// TwinCAT 3 PLC project ExampleProject
// ProgramVersion: 3.1.4026.9
// CompilerDefines: VISU_USEWSTRING
// libraries:
//   Tc2_Standard, * (Beckhoff Automation GmbH)
//   Tc2_System, * (Beckhoff Automation GmbH)
//   Core, * (_)
//   Utils, * (_)
// project tree:
//   / GlobalTextList.TcGTLO, PlcTask.TcTTO
//   Heating/Ctx/ Heating_Ctx_Hmi.TcPOU, Heating_Ctx_Io.TcDUT, Heating_Ctx_Priv.TcPOU, Heating_Ctx_States.TcPOU (not stored)
//   Heating/Ctx/Io/ Heating_Ctx_Io_In.TcDUT (not stored), Heating_Ctx_Io_Out.TcDUT (not stored)
//   Heating/ Heating.TcPOU, Heating_Ctx.TcPOU
//   Heating/Receivers/ Heating_PassiveCountRec.TcPOU, Heating_RequestRec.TcPOU
//   Heating/State/ Heating_State.TcPOU (not stored), Heating_State_Enabled.TcPOU, Heating_State_Disabled.TcPOU, Heating_State_Heatup.TcPOU, Heating_State_Pumping.TcPOU, Heating_State_Safety.TcPOU, Heating_State_Fault.TcPOU
//   MAIN/ ArgAsIRoom.TcPOU, CST.TcGVL, COL.TcGVL, MAIN.TcPOU
//   Room/Rooms/FullRoom/ PassiveTempTimeRoomWithMultipleValves.TcPOU, Room_Settings_PassiveTempTime.TcDUT (not stored), PassiveTempTimeRoom.TcPOU
//   Room/Rooms/PassiveRoom/ PassiveRoom.TcPOU
//   Room/Rooms/TempRoom/ Room_Settings_TemperatureSettings.TcDUT, TempRoom.TcPOU, TempRoomWithMultipleSensors.TcPOU
//   Room/Rooms/TimeRoom/ Room_Settings_TimeSettings.TcDUT, TimeRoom.TcPOU
//   Room/Rooms/TempTimeRoom/ Room_Settings_TempTime.TcDUT (not stored), TempTimeRoom.TcPOU
//   Room/Shared Interface/ I_Room.TcIO, RoomInterface.TcPOU (not stored)
//   Room/Ctx/ Room_Ctx_Hmi.TcPOU, Room_Ctx_Io.TcDUT, Room_Ctx_Priv.TcPOU, Room_Ctx_States.TcPOU
//   Room/Receivers/ Room_SystemReceiver.TcPOU
//   Room/Rooms/ AbstractRoom.TcPOU
//   Room/ Room_Ctx.TcPOU
//   Room/State/ Room_State.TcPOU, Room_State_DemandPassive.TcPOU, Room_State_Idle.TcPOU, Room_State_Fault.TcPOU, Room_State_DemandTemperature.TcPOU, Room_State_Disabled.TcPOU, Room_State_DemandTime.TcPOU, Room_State_SystemOff.TcPOU
//   Room/UI/ Room_UiLogic.TcPOU
//   Safety/ Safety.TcPOU, Safety_Hmi.TcPOU

CONFIGURATION ExampleProject
    RESOURCE PLC ON TwinCAT3
        TASK PlcTask(INTERVAL := T#10ms, PRIORITY := 20);
        PROGRAM MAIN WITH PlcTask : MAIN;
    END_RESOURCE
END_CONFIGURATION

// ---- Heating/Ctx/Heating_Ctx_Io.TcDUT
TYPE Heating_Ctx_Io :
STRUCT
	in		: Heating_Ctx_Io_In;
	out		: Heating_Ctx_Io_Out;
END_STRUCT
END_TYPE

// ---- Room/Rooms/TempRoom/Room_Settings_TemperatureSettings.TcDUT
TYPE Room_Settings_TemperatureSettings :
STRUCT
	rLow	: REAL := 19.0;
	rHigh	: REAL := 19.3;
END_STRUCT
END_TYPE

// ---- Room/Rooms/TimeRoom/Room_Settings_TimeSettings.TcDUT
TYPE Room_Settings_TimeSettings :
STRUCT
	nOff		: UDINT := TIME_TO_UDINT(T#30S);
	nOn			: UDINT := TIME_TO_UDINT(T#30S);
END_STRUCT
END_TYPE

// ---- Room/Ctx/Room_Ctx_Io.TcDUT
TYPE Room_Ctx_Io :
STRUCT
	in		: Heating_Ctx_Io_In;
	out		: Heating_Ctx_Io_Out;
END_STRUCT
END_TYPE

// ---- MAIN/CST.TcGVL
{attribute 'qualified_only'}
VAR_GLOBAL CONSTANT
	MAX_PASSIVE_ROOM		: UDINT := 3;
END_VAR

// ---- MAIN/COL.TcGVL
{attribute 'qualified_only'}
VAR_GLOBAL CONSTANT
{warning disable C0228}	// Disable warning: No initial value for variable ...
	RED			: Color(255, 0, 0, 255);
	BLACK		: Color(0, 0, 0, 255);
	ORANGE		: Color(255, 160, 0, 255);
	WHITE		: Color(255, 255, 255, 255);
{warning restore C0228}
END_VAR

// ---- Room/Shared Interface/I_Room.TcIO
INTERFACE I_Room EXTENDS I_Arg

PROPERTY Active : BOOL
GET
END_GET
END_PROPERTY

METHOD Close
END_METHOD

PROPERTY Id : UDINT
GET
END_GET
END_PROPERTY

PROPERTY IsClosed : BOOL
GET
END_GET
END_PROPERTY

PROPERTY IsOpen : BOOL
GET
END_GET
END_PROPERTY

PROPERTY IsReady : BOOL
GET
END_GET
END_PROPERTY

METHOD Open
END_METHOD

PROPERTY Timeout : TIME
GET
END_GET
END_PROPERTY

METHOD TriggerFault
VAR_INPUT
	sErrorText		: Str;
END_VAR
END_METHOD

END_INTERFACE

// ---- MAIN/MAIN.TcPOU
PROGRAM MAIN
VAR
	safety				: Safety<2>;
	heating				: Heating;
	standardRoom		: ARRAY[1..5] OF TempTimeRoom;
	receptionRoom		: PassiveRoom;
	conferentionRoom01	: PassiveTempTimeRoom;
	conferentionRoom02	: PassiveTempTimeRoomWithMultipleValves<3>;
	storeRoom01			: TempRoom;
	storeRoom02			: TempRoomWithMultipleSensors<3>;
	
	bSimulation			: BOOL;
	
	dbgList				: DebugList;	
	
	
	
END_VAR

Runtime();

IF bSimulation THEN
	_Sim();
ELSE
	_IO();	
END_IF

METHOD PRIVATE _IO
END_METHOD

METHOD PRIVATE _Sim
IF safety.bErrAck THEN
	safety.bSafetyOk := TRUE;
END_IF
END_METHOD

END_PROGRAM

// ---- Safety/Safety.TcPOU
FUNCTION_BLOCK Safety 
VAR_GENERIC CONSTANT
	ESTOP_CAP		: UDINT := 2;
END_VAR
IMPLEMENTS I_Execute
VAR_INPUT
	bSafetyOk		: BOOL;
	bEStopActive	: ARRAY[1..ESTOP_CAP] OF BOOL;
END_VAR
VAR_OUTPUT
	bSafetyRun		: BOOL;
	bErrAck			: BOOL;
END_VAR
VAR
	_this			: Entity;
	_ctx			: Heating_Ctx;
	_tag			: Tag('Safety');
	_compTag		: Comp(_tag, _this);
	_exe			: Execute(THIS^);
	
	_onSafetyChange		: Signal;
	_compOnSafetyChange	: Comp(_onSafetyChange, _this);
	
	_bSafetyStopActive	: BoolArg;
	
	_hmi				: Safety_Hmi<ESTOP_CAP>;
	
	_nStep				: USINT;
	_tonTimeout			: TON;
END_VAR

METHOD Execute
VAR
	i			: UDINT;
END_VAR
FOR i := 1 TO ESTOP_CAP DO
	_hmi.bEStopActive[i] := bESTopActive[i];
END_FOR


CASE _nStep OF
	0: // Fault Init
		_bSafetyStopActive.Val := TRUE;
		_onSafetyChange.Emit(_bSafetyStopActive);
		bSafetyRun	:= FALSE;
		
		_nStep := 1;
		
		_hmi.bHideReset := FALSE;
		_hmi.nStatusColor := COL.RED.Raw;
		_hmi.sStatusText := 'Safety Stop Activated!';

	1: // Fault
		IF bSafetyOk AND _hmi.bReset THEN
			_hmi.bReset := FALSE;
			
			_nStep := 2;
		END_IF

	2: // Reset init
		bSafetyRun	:= TRUE;
		
		_nStep		:= 3;
		
		_hmi.bHideReset := FALSE;
		_hmi.nStatusColor := COL.RED.Raw;
		_hmi.sStatusText := 'Reset in progress...';
		
	3: // Reset
	
		bErrAck		:= TRUE;
		
		_tonTimeout(IN := TRUE, PT := T#5S);
		
		IF bSafetyOk THEN
			_tonTimeout(IN := FALSE);
			_nStep := 4;
		ELSIF _tonTimeout.Q THEN
			_tonTimeout(IN := FALSE);
			_nStep := 0;
		END_IF	

	4:	// Op Init
		bErrAck		:= FALSE;
	
		_bSafetyStopActive.Val := FALSE;
		_onSafetyChange.Emit(_bSafetyStopActive);
		_nStep := 5;
		
		_hmi.bHideReset := FALSE;
		_hmi.nStatusColor := COL.BLACK.Raw;
		_hmi.sStatusText := 'Safety OK!';

	5:	// Op
		IF NOT bSafetyOk THEN
			_nStep := 0;
		END_IF


		
END_CASE
END_METHOD

END_FUNCTION_BLOCK

// ---- Heating/Heating_Ctx.TcPOU
FUNCTION_BLOCK Heating_Ctx
VAR_INPUT
	io		: Heating_Ctx_Io;
	hmi		: Heating_Ctx_Hmi;
	state	: Heating_Ctx_States;
	priv	: Heating_Ctx_Priv;
END_VAR

END_FUNCTION_BLOCK

// ---- Heating/Ctx/Heating_Ctx_Hmi.TcPOU
FUNCTION_BLOCK Heating_Ctx_Hmi
VAR_INPUT
	sStatusText				: Str;
	nStatusColor			: LWORD;
	
	bButton					: BOOL;
	sButtonText				: Str;
	nButtonColor			: LWORD;	
END_VAR

END_FUNCTION_BLOCK

// ---- Heating/Ctx/Heating_Ctx_Priv.TcPOU
FUNCTION_BLOCK Heating_Ctx_Priv
VAR_INPUT
	iActiveRoom		: I_Arg;
	nPassiveRooms	: UDINT;	
END_VAR
VAR_OUTPUT
	iOnEnable		: I_SignalEmit;
	iOnDisable		: I_SignalEmit;
	iOnPause		: I_SignalEmit;
	iOnResume		: I_SignalEmit;
	
	iQueue			: I_MutArgQueue;
END_VAR

END_FUNCTION_BLOCK

// ---- Safety/Safety_Hmi.TcPOU
FUNCTION_BLOCK Safety_Hmi
VAR_GENERIC CONSTANT
	ESTOP_CAP		: UDINT := 4;
END_VAR

VAR_INPUT
	bEStopActive	: ARRAY[1..ESTOP_CAP] OF BOOL;
	
	sStatusText		: Str;
	nStatusColor	: LWORD;
	
	bReset			: BOOL;
	bHideReset		: BOOL;
END_VAR

END_FUNCTION_BLOCK

// ---- Heating/Heating.TcPOU
FUNCTION_BLOCK Heating IMPLEMENTS I_Execute
VAR_INPUT
	bPumpOverload	: BOOL;
	bBurnerOverload	: BOOL;

	rBoilerTemp		: REAL;
	rBoilerPressure	: REAL;	
END_VAR
VAR_OUTPUT
	bPump			: BOOL;
	bBurner			: BOOL;
END_VAR
VAR
	_this			: Entity;
	_ctx			: Heating_Ctx;
	_tag			: Tag('Heating');
	_compTag		: Comp(_tag, _this);
	_exe			: Execute(THIS^);
	
	_onEnable		: Signal;
	_compOnEnable	: Comp(_onEnable, _this);
	_proxOnEnable	: SignalProxy(_onEnable, _ctx.priv.iOnEnable);
	
	_onDisable		: Signal;
	_compOnDisable	: Comp(_onDisable, _this);
	_proxOnDisable	: SignalProxy(_onDisable, _ctx.priv.iOnDisable);
	
	_onPause		: Signal;
	_compOnPause	: Comp(_onPause, _this);
	_proxOnPause	: SignalProxy(_onPause, _ctx.priv.iOnPause);
	
	_onResume		: Signal;
	_compOnResume	: Comp(_onResume, _this);
	_proxOnResume	: SignalProxy(_onResume, _ctx.priv.iOnResume);
	
	_smgr			: StateManager<6>(_this);
	_proxSmgr		: StateManagerProxy(_smgr, _ctx.state.iMgr);
	
	_disabled		: Heating_State_Disabled(_this, _ctx);
	_proxDisabled	: StateProxy(_disabled, _ctx.state.iDisable);
	
	_safety			: Heating_State_Safety(_this, _ctx);
	_proxSafety		: StateProxy(_safety, _ctx.state.iSafety);
	
	_fault			: Heating_State_Fault(_this, _ctx);
	_proxFault		: StateProxy(_fault, _ctx.state.iFault);
	
	_enabled		: Heating_State_Enabled(_this, _ctx);
	_proxEnabled	: StateProxy(_enabled, _ctx.state.iEnable);
	
	_pumping		: Heating_State_Pumping(_this, _ctx);
	_proxPumping	: StateProxy(_pumping, _ctx.state.iPump);
	
	_heatup			: Heating_State_Heatup(_this, _ctx);
	_proxHeatup		: StateProxy(_heatup, _ctx.state.iHeatup);

	_passiveHeatingCount		: Heating_PassiveCountRec(_ctx);
	_passiveHeatingCountRec		: Receiver(_passiveHeatingCount);
	_compPassiveHeatingCountRec	: Comp(_passiveHeatingCountRec, _this);
	
	_request					: Heating_RequestRec(_ctx);
	_requestRec					: Receiver(_request);
	_compRequestRec				: Comp(_requestRec, _this);
	
	_queue						: ArgQueue<CST.MAX_ROOM>;
	_queueProxy					: ArgQueueProxy(_queue, _ctx.priv.iQueue);
	
	_tonPump	: TON;
	_tonBurner	: TON;
END_VAR

METHOD Execute
// Inputs
_ctx.io.in.bBurnerOverload := bBurnerOverload;
_ctx.io.in.bPumpOverload := bPumpOverload;
_ctx.io.in.rBoilerPressure := rBoilerPressure;
_ctx.io.in.rBoilerTemp := rBoilerTemp;

// Outputs
_tonPump(IN := _ctx.io.out.bPump, PT := T#2S, Q => bPump);
_tonBurner(IN := _ctx.io.out.bBurner, PT := T#2S, Q => bBurner);
END_METHOD

END_FUNCTION_BLOCK

// ---- Heating/State/Heating_State_Disabled.TcPOU
FUNCTION_BLOCK Heating_State_Disabled EXTENDS Heating_State
VAR_INPUT
END_VAR
VAR_OUTPUT
END_VAR
VAR
END_VAR

METHOD OnExecute
IF _ctx.hmi.bButton THEN
	_ctx.hmi.bButton := FALSE;
	_ctx.state.iMgr.Request(_ctx.state.iEnable);
END_IF
END_METHOD

METHOD OnInit
_ctx.hmi.sStatusText := 'Heating disabled!';
_ctx.hmi.nStatusColor := COL.BLACK.Raw;

_ctx.hmi.sButtonText := 'Press to ENABLE!';
_ctx.hmi.nButtonColor := COL.BLACK.Raw;

_ctx.io.out.bBurner := FALSE;
_ctx.io.out.bPump := FALSE;

_ctx.priv.iOnDisable.Emit();
END_METHOD

END_FUNCTION_BLOCK

// ---- Heating/State/Heating_State_Safety.TcPOU
FUNCTION_BLOCK Heating_State_Safety EXTENDS Heating_State IMPLEMENTS I_Callable, I_Init
VAR
	_init					: Init(THIS^);
	_safetyRec				: Receiver(THIS^);
	_bSafetyStopActive			: BOOL;
END_VAR

METHOD Call
VAR_INPUT
	iArg		: Core.I_Arg;
END_VAR
VAR
	_iSafeModeOn: I_BoolArg;
END_VAR
IF IsOk(ArgToIBoolArg(iArg, iVal => _iSafeModeOn)) THEN
	IF _iSafeModeOn.Val THEN
		_bSafetyStopActive := TRUE;
		_ctx.state.iMgr.Request(_ctx.state.iSafety);
	ELSE
		_bSafetyStopActive := FALSE;
		_ctx.state.iMgr.Request(_ctx.state.iDisable);
	END_IF
END_IF
END_METHOD

METHOD CanDeactivate : BOOL
CanDeactivate := NOT _bSafetyStopActive;
END_METHOD

METHOD Init
VAR
	i			: Iter(1);
	_r			: Result;
	
	_iEntity	: I_Entity;
	_iSignal	: I_Signal;
	
	
END_VAR
WHILE IsOk(GetEntity(i.Next(), iEntity => _iEntity)) DO
	IF IsOk(GetSignal(_iEntity, '*.onSafetyChange', iSignal => _iSignal)) THEN
		IF IsErr(_iSignal.Pair(_safetyRec), nOut => _r) THEN
			DebugMsg(_iSignal, CONCAT('Could not be paired! Error code: ', TO_STRING(_r)));
		END_IF
		
		EXIT;
	END_IF
END_WHILE

IF NOT IsOk(_r) THEN
	DebugMsg(THIS^, CONCAT('_safetyRec not paired! Error code: ', TO_STRING(_r)));
END_IF
END_METHOD

METHOD OnInit
_ctx.hmi.sStatusText := 'Safety engaged! Check safety system...';
_ctx.hmi.nStatusColor := COL.RED.Raw;

_ctx.hmi.sButtonText := '';
_ctx.hmi.nButtonColor := COL.INVISIBLE.Raw;

_ctx.io.out.bBurner := FALSE;
_ctx.io.out.bPump := FALSE;

_ctx.priv.iOnDisable.Emit();
END_METHOD

END_FUNCTION_BLOCK

// ---- Heating/State/Heating_State_Fault.TcPOU
FUNCTION_BLOCK Heating_State_Fault EXTENDS Heating_State
VAR_INPUT
END_VAR
VAR_OUTPUT
END_VAR
VAR
END_VAR

METHOD OnInit
_ctx.hmi.sStatusText := 'Heating enabled: Waiting for requests...';
_ctx.hmi.nStatusColor := COL.BLACK.Raw;

_ctx.hmi.sButtonText := 'Press to DISABLE!';
_ctx.hmi.nButtonColor := COL.BLACK.Raw;

_ctx.io.out.bBurner := FALSE;
_ctx.io.out.bPump := FALSE;
END_METHOD

END_FUNCTION_BLOCK

// ---- Heating/State/Heating_State_Enabled.TcPOU
FUNCTION_BLOCK Heating_State_Enabled EXTENDS Heating_State
VAR_INPUT
END_VAR
VAR_OUTPUT
END_VAR
VAR
END_VAR

METHOD OnExecute
VAR
	_iRoomArg		: I_Arg;
END_VAR
IF _ctx.hmi.bButton THEN
	_ctx.hmi.bButton := FALSE;
	_ctx.state.iMgr.Request(_ctx.state.iDisable);
	
ELSIF _ctx.io.in.rBoilerTemp < _ctx.hmi.rMinTemperature THEN
	_ctx.state.iMgr.Request(_ctx.state.iHeatup);
	
ELSIF IsOk(_ctx.priv.iQueue.Pop(iArg => _iRoomArg)) THEN
	IF IsOk(ArgAsIRoom(_iRoomArg, iDest => _ctx.priv.iActiveRoom)) THEN
		_ctx.state.iMgr.Request(_ctx.state.iPump);
	ELSE
		_ctx.hmi.sErrorText := 'Room Queue - Incorrect iRoomArg!';
	END_IF
END_IF

IF NOT _ctx.io.out.bPump AND _ctx.priv.nPassiveRooms <> 0 THEN
	_ctx.io.out.bPump := TRUE;
	_ctx.hmi.sStatusText := 'Heating enabled: Circulating...';
	
ELSIF _ctx.io.out.bPump AND _ctx.priv.nPassiveRooms <> 0 THEN
	_ctx.io.out.bPump := FALSE;
	_ctx.hmi.sStatusText := 'Heating enabled: Waiting for requests...';
	
END_IF
END_METHOD

METHOD OnInit
_ctx.hmi.sStatusText := 'Heating enabled: Waiting for requests...';
_ctx.hmi.nStatusColor := COL.BLACK.Raw;

_ctx.hmi.sButtonText := 'Press to DISABLE!';
_ctx.hmi.nButtonColor := COL.BLACK.Raw;

_ctx.io.out.bBurner := FALSE;
_ctx.io.out.bPump := FALSE;

_ctx.priv.iOnEnable.Emit();
_ctx.priv.iOnResume.Emit();
END_METHOD

END_FUNCTION_BLOCK

// ---- MAIN/ArgAsIRoom.TcPOU
FUNCTION ArgAsIRoom : Result
VAR_INPUT
	iSource	: I_Arg;
END_VAR
VAR_OUTPUT
	iDest	: I_Room;
END_VAR

IF iSource = 0 THEN
	ArgAsIRoom := Err.Itf0;
	RETURN;
END_IF

IF __QUERYINTERFACE(iSource, iDest) THEN
	ArgAsIRoom := Ok;
ELSE
	ArgAsIRoom := Err.NoMatch;
END_IF

END_FUNCTION

// ---- Heating/State/Heating_State_Pumping.TcPOU
FUNCTION_BLOCK Heating_State_Pumping EXTENDS Heating_State
VAR CONSTANT
	ERROR_STEP		: USINT := 8;
	READY_STEP		: USINT := 9;
END_VAR
VAR
	_nStep		: USINT;
	_tonTimeout	: TON;
END_VAR

METHOD CanActivate : BOOL
CanActivate :=  _ctx.state.iMgr.Current = _ctx.state.iEnable;
END_METHOD

METHOD OnExecute
VAR
	strb		: Strb;
END_VAR
_tonTimeout(IN := TRUE);
IF _tonTimeout.Q THEN
	_nStep := ERROR_STEP;
	_ctx.hmi.sErrorText := strb.Append('Pumping - Timeout at step ')
								.Append(USINT_TO_STRING(_nStep))
								.Append('!')
								.Read();
ELSIF _ctx.priv.iActiveRoom = 0 THEN
	_nStep := ERROR_STEP;
	_ctx.hmi.sErrorText := 'Pumping -Incorrect iActiveRoom value!';
ELSIF _ctx.priv.iActiveRoom.Abort THEN
	_nStep := 6;
END_IF

CASE _nStep OF
	0:
		_ctx.priv.iActiveRoom.Open();
		_nStep := 1;
		
	1:
		IF _ctx.priv.iActiveRoom.IsOpen THEN
			_nStep := 2;
		END_IF
	2:	
		_ctx.io.out.bBurner := TRUE;
		_ctx.io.out.bPump := TRUE;
		_nStep := 3;
		
	3:
		_tonTimeout(IN := FALSE);
		IF _ctx.priv.iActiveRoom.IsReady THEN
			_nStep := 4;
		END_IF
	4:	
		_ctx.io.out.bBurner := FALSE;
		_ctx.io.out.bPump := FALSE;
		_nStep := 5;
	5:
		_ctx.priv.iActiveRoom.Close();
		_nStep := 6;
	6:
		IF _ctx.priv.iActiveRoom.IsClosed THEN
			_nStep := 7;
		END_IF
	7:
		_ctx.state.iMgr.Request(_ctx.state.iEnable);
		_nStep := READY_STEP;
	ERROR_STEP:
		_ctx.state.iMgr.Request(_ctx.state.iFault);
		_nStep := READY_STEP;
END_CASE
END_METHOD

METHOD OnInit
VAR
	strb			: Strb;
END_VAR
_ctx.hmi.sStatusText := strb.Append('Heating enabled: Pumping to room ')
							.Append(UDINT_TO_STRING(_ctx.priv.iActiveRoom.Id))
							.Append('...')
							.Read();
							
_ctx.hmi.nStatusColor := COL.BLACK.Raw;

_ctx.hmi.sButtonText := 'Press to DISABLE!';
_ctx.hmi.nButtonColor := COL.BLACK.Raw;

_ctx.io.out.bBurner := FALSE;
_ctx.io.out.bPump := FALSE;

_ctx.priv.iOnPause.Emit();

_nStep := 0;
_tonTimeout(IN := FALSE);
END_METHOD

END_FUNCTION_BLOCK

// ---- Heating/State/Heating_State_Heatup.TcPOU
FUNCTION_BLOCK Heating_State_Heatup EXTENDS Heating_State
VAR_INPUT
END_VAR
VAR_OUTPUT
END_VAR
VAR
END_VAR

METHOD CanActivate : BOOL
CanActivate :=  _ctx.state.iMgr.Current = _ctx.state.iEnable;
END_METHOD

METHOD OnExecute
IF _ctx.hmi.bButton THEN
	_ctx.hmi.bButton := FALSE;
	_ctx.state.iMgr.Request(_ctx.state.iEnable);
END_IF
END_METHOD

METHOD OnInit
_ctx.hmi.sStatusText := 'Heating enabled: Heating up...';
_ctx.hmi.nStatusColor := COL.BLACK.Raw;

_ctx.hmi.sButtonText := 'Press to DISABLE!';
_ctx.hmi.nButtonColor := COL.BLACK.Raw;

_ctx.io.out.bBurner := TRUE;
_ctx.io.out.bPump := TRUE;
END_METHOD

END_FUNCTION_BLOCK

// ---- Heating/Receivers/Heating_PassiveCountRec.TcPOU
FUNCTION_BLOCK Heating_PassiveCountRec IMPLEMENTS I_Callable
VAR
	_ctx			: REFERENCE TO Heating_Ctx;
END_VAR

METHOD Call
VAR_INPUT
	iArg				: Core.I_Arg;
END_VAR
VAR
	_iPassiveHeatingOn	: I_BoolArg;
END_VAR
IF IsOk(ArgToIBoolArg(iArg, iVal => _iPassiveHeatingOn)) THEN
	IF _iPassiveHeatingOn.Val THEN
		IF _ctx.priv.nPassiveRooms > CST.MAX_PASSIVE_ROOM THEN
			_ctx.priv.nPassiveRooms := _ctx.priv.nPassiveRooms + 1;
		END_IF 	
	ELSE
		IF _ctx.priv.nPassiveRooms > 0 THEN
			_ctx.priv.nPassiveRooms := _ctx.priv.nPassiveRooms - 1;
		END_IF
	END_IF
END_IF
END_METHOD

//FB_Init is always available implicitly and it is used primarily for initialization.
//The return value is not evaluated. For a specific influence, you can also declare the
//methods explicitly and provide additional code there with the standard initialization
//code. You can evaluate the return value.
METHOD FB_Init: BOOL
VAR_INPUT
    bInitRetains: BOOL; // TRUE: the retain variables are initialized (reset warm / reset cold)
    bInCopyCode: BOOL;  // TRUE: the instance will be copied to the copy code afterward (online change)

	ctx			: REFERENCE TO Heating_Ctx;   
END_VAR
_ctx REF= ctx;
END_METHOD

END_FUNCTION_BLOCK

// ---- Heating/Receivers/Heating_RequestRec.TcPOU
FUNCTION_BLOCK Heating_RequestRec IMPLEMENTS I_Callable
VAR
	_ctx			: REFERENCE TO Heating_Ctx;
END_VAR

METHOD Call
VAR_INPUT
	iArg				: Core.I_Arg;
END_VAR
VAR
	_iRoom				: I_Room;
END_VAR
IF IsOk(ArgAsIRoom(iArg, iDest => _iRoom)) THEN
	_ctx.priv.iQueue.Push(_iRoom);
END_IF
END_METHOD

//FB_Init is always available implicitly and it is used primarily for initialization.
//The return value is not evaluated. For a specific influence, you can also declare the
//methods explicitly and provide additional code there with the standard initialization
//code. You can evaluate the return value.
METHOD FB_Init: BOOL
VAR_INPUT
    bInitRetains: BOOL; // TRUE: the retain variables are initialized (reset warm / reset cold)
    bInCopyCode: BOOL;  // TRUE: the instance will be copied to the copy code afterward (online change)

	ctx			: REFERENCE TO Heating_Ctx;   
END_VAR
_ctx REF= ctx;
END_METHOD

END_FUNCTION_BLOCK

// ---- Room/Rooms/TempTimeRoom/TempTimeRoom.TcPOU
FUNCTION_BLOCK TempTimeRoom IMPLEMENTS I_Execute
VAR CONSTANT
	STATE_CAP		: UDINT := 6;
END_VAR
VAR
	_this			: Entity;
	_ctx			: Room_Ctx;
	_room			: RoomInterface(_ctx);
	_tag			: Tag(CONCAT('Room_', UDINT_TO_STRING(_room.Id)));
	_compTag		: Comp(_tag, _this);
	_exe			: Execute(THIS^);
	
	_uiLogic		: Room_UiLogic(_ctx);
	
	_systemReceiver	: Room_SystemReceiver(_ctx);
	
	_smgr			: StateManager<STATE_CAP>(_this);
	_proxSmgr		: StateManagerProxy(_smgr, _ctx.state.iMgr);
	
	_disable		: Room_State_Disabled(_this, _ctx);
	_proxDisable	: StateProxy(_disable, _ctx.state.iDisable);
	
	_fault			: Room_State_Fault(_this,_ctx);
	_proxFault		: StateProxy(_fault, _ctx.state.iFault);	
	
	_idle			: Room_State_Idle(_this,_ctx);
	_proxIdle		: StateProxy(_idle, _ctx.state.iIdle);	
	
	_systemOff		: Room_State_SystemOff(_this,_ctx);
	_proxSystemOff	: StateProxy(_systemOff, _ctx.state.iSystemOff);
END_VAR

// Here add custom components

VAR PERSISTENT
	_settings		: Room_Settings_TempTime;
END_VAR

VAR_INPUT
	rTemperature	: REAL;
	
	bInletValveIsOpen		: BOOL;
	bInletValveIsClosed		: BOOL;
	
	bOutletValveIsOpen		: BOOL;
	bOutletValveIsClosed	: BOOL;
END_VAR
VAR_OUTPUT
	bInletValve			: BOOL;
	bOutletValve		: BOOL;
END_VAR

VAR
	_timeDemand		: Room_State_DemandTime(_this, _ctx, _settings.timee);
	_tempDemand		: Room_State_DemandTemperature(_this, _ctx, _settings.temp, rTemperature);
END_VAR

METHOD Execute
_ctx.priv.bClosed := bInletValveIsClosed AND bOutletValveIsClosed;
_ctx.priv.bOpen := bInletValveIsOpen AND bOutletValveIsOpen;

bInletValve :=  _ctx.io.bOpenValves;
bOutletValve :=  _ctx.io.bOpenValves;
END_METHOD

END_FUNCTION_BLOCK

// ---- Room/Room_Ctx.TcPOU
FUNCTION_BLOCK Room_Ctx
VAR_INPUT
	io		: Room_Ctx_Io;
	hmi		: Room_Ctx_Hmi;
	state	: Room_Ctx_States;
	priv	: Room_Ctx_Priv;
END_VAR

END_FUNCTION_BLOCK

// ---- Room/Ctx/Room_Ctx_Hmi.TcPOU
FUNCTION_BLOCK Room_Ctx_Hmi
VAR_INPUT
	sStatusText				: Str;
	sErrorText				: Str;
	nStatusColor			: LWORD;
	
	sData					: Str;
	
	bDisable				: BOOL;
	sDisableText			: Str;
	
	bReset					: BOOL;
	bHideReset				: BOOL;
END_VAR
VAR_OUTPUT PERSISTENT
	nTimeout				: UDINT := TIME_TO_UDINT(T#60S);
END_VAR

END_FUNCTION_BLOCK

// ---- Room/Ctx/Room_Ctx_States.TcPOU
FUNCTION_BLOCK Room_Ctx_States
VAR_OUTPUT
	iMgr			: I_StateManager;
	
	iSafety			: I_State;
	iFault			: I_State;
	iDisable		: I_State;
	iEnable			: I_State;
	iPump			: I_State;
	iHeatup			: I_State;
	
END_VAR

END_FUNCTION_BLOCK

// ---- Room/Ctx/Room_Ctx_Priv.TcPOU
FUNCTION_BLOCK Room_Ctx_Priv
VAR_INPUT
	bReady		: BOOL;
	bOpen		: BOOL;
	bClosed		: BOOL;
	bActive		: BOOL;
	
	bPaused		: BOOL;
	bSysOff		: BOOL;
	
	iThisRoom	: I_Room;
END_VAR

END_FUNCTION_BLOCK

// ---- Room/UI/Room_UiLogic.TcPOU
FUNCTION_BLOCK Room_UiLogic IMPLEMENTS I_Execute
VAR_INPUT
END_VAR
VAR_OUTPUT
END_VAR
VAR
	_exe			: Execute(THIS^);
	_ctx			: REFERENCE TO Room_Ctx;
	
	_bPrvDisable	: BOOL;
END_VAR

METHOD Execute
IF _bPrvDisable <> _ctx.hmi.bDisable THEN
	_bPrvDisable := _ctx.hmi.bDisable;
	
	IF _ctx.hmi.bDisable THEN
		_ctx.hmi.sDisableText := 'Press to ENABLE!';
	ELSE
		_ctx.hmi.sDisableText := 'Press to DISABLE!';
	END_IF	
END_IF
END_METHOD

//FB_Init is always available implicitly and it is used primarily for initialization.
//The return value is not evaluated. For a specific influence, you can also declare the
//methods explicitly and provide additional code there with the standard initialization
//code. You can evaluate the return value.
METHOD FB_Init: BOOL
VAR_INPUT
    bInitRetains: BOOL; // TRUE: the retain variables are initialized (reset warm / reset cold)
    bInCopyCode: BOOL;  // TRUE: the instance will be copied to the copy code afterward (online change)
	
	ctx			: REFERENCE TO Room_Ctx;
END_VAR
_ctx REF= ctx;
END_METHOD

END_FUNCTION_BLOCK

// ---- Room/Receivers/Room_SystemReceiver.TcPOU
FUNCTION_BLOCK Room_SystemReceiver IMPLEMENTS I_Init, I_Callable
VAR
	_init			: Init(THIS^);
	_systemRec		: Receiver(THIS^);
	
	_bError			: BOOL;
	
	_iOnResume		: I_Signal;
	_iOnPause		: I_Signal;
	_iOnEnable		: I_Signal;
	_iOnDisable		: I_Signal;
	
	_ctx			: REFERENCE TO Room_Ctx;
	
	_iOnPauseBehaviour	: I_Callable;
	_iOnResumeBehaviour	: I_Callable;
END_VAR

METHOD PRIVATE _GetSignalAndPair
VAR_INPUT
	iEntity		: I_Entity;
	sToFind		: Str;
END_VAR
VAR_OUTPUT
	iSignal	: I_Signal;
END_VAR
VAR
	_r			: Result;
	strb		: Strb;
END_VAR
CASE GetSignal(iEntity, sToFind, iSignal => iSignal) OF
	Ok:
		IF IsErr(iSignal.Pair(_systemRec), nOut => _r) THEN
			_bError := TRUE;
			DebugMsg(iSignal, strb.Append('Cannot pair _systemRec with this signal! Error code: ').Append(TO_STRING(_r)).Read());
		END_IF
	ELSE
		_bError := TRUE;
		DebugMsg(THIS^, strb.Append('Cannot pair _systemRec with a ').Append(sToFind).Append('!').Read());
		DebugMsg(iEntity, strb.Append(sToFind).Append(' not found!').Read());
END_CASE
END_METHOD

METHOD Call
VAR_INPUT
	iArg	: Core.I_Arg;
END_VAR
VAR
	cmp		: TagCmp;
	cmp2	: TagCmp;
	_iTag	: I_Tag;
END_VAR
IF _bError THEN
	_ctx.hmi.sErrorText := 'Incorrect receiver initialization!';
	_ctx.state.iMgr.Request(_ctx.state.iFault);
	RETURN;
END_IF

IF IsErr(ArgAsITag(iArg, iDest => _iTag)) THEN
	_ctx.hmi.sErrorText := 'Incorrect call argument!';
	_ctx.state.iMgr.Request(_ctx.state.iFault);
	RETURN;
END_IF

cmp.Set(_iTag);
cmp2.Set(_ctx.state.iMgr.Current.Tag);
IF cmp.Match(_iOnResume.Tag).IsTrue() THEN
	_ctx.priv.bPaused := FALSE;		
	RETURN;
END_IF

IF cmp.Match(_iOnPause.Tag).IsTrue() THEN
	_ctx.priv.bPaused := TRUE;
	RETURN;
END_IF

IF cmp.Match(_iOnEnable.Tag).IsTrue() THEN
	IF cmp2.Match(_ctx.state.iSystemOff.Tag).IsFalse() THEN
		RETURN;
	END_IF
	
	IF cmp2.Match(_ctx.state.iIdle.Tag).IsTrue() THEN
		RETURN;
	END_IF
	_ctx.priv.bSysOff := FALSE;
	_ctx.state.iMgr.Request(_ctx.state.iIdle);	
	RETURN;
END_IF

IF cmp.Match(_iOnDisable.Tag).IsTrue() THEN
	IF cmp2.Match(_ctx.state.iSystemOff.Tag).IsTrue() THEN
		RETURN;
	END_IF	
	_ctx.priv.bSysOff := TRUE;
	_ctx.state.iMgr.Request(_ctx.state.iSystemOff);
	RETURN;
END_IF
END_METHOD

//FB_Init is always available implicitly and it is used primarily for initialization.
//The return value is not evaluated. For a specific influence, you can also declare the
//methods explicitly and provide additional code there with the standard initialization
//code. You can evaluate the return value.
METHOD FB_Init: BOOL
VAR_INPUT
    bInitRetains: BOOL; // TRUE: the retain variables are initialized (reset warm / reset cold)
    bInCopyCode: BOOL;  // TRUE: the instance will be copied to the copy code afterward (online change)
	
	ctx			: REFERENCE TO Room_Ctx;
END_VAR
_ctx REF= ctx;
END_METHOD

METHOD Init
VAR
	i			: Iter(1);
	_iEntity	: I_Entity;
END_VAR
WHILE IsOk(GetEntity(i.Next(), iEntity => _iEntity)) DO
	IF IsNone(GetTagOpt(_iEntity, 'Heating')) THEN
		CONTINUE;
	END_IF
	
	_GetSignalAndPair(_iEntity, '*._onPause', iSignal => _iOnPause);
	_GetSignalAndPair(_iEntity, '*._onResume', iSignal => _iOnResume);
	_GetSignalAndPair(_iEntity, '*._onEnable', iSignal => _iOnEnable);
	_GetSignalAndPair(_iEntity, '*._onDisable', iSignal => _iOnDisable);
END_WHILE
END_METHOD

END_FUNCTION_BLOCK

// ---- Room/State/Room_State_Disabled.TcPOU
FUNCTION_BLOCK Room_State_Disabled EXTENDS Room_State
VAR_INPUT
END_VAR
VAR_OUTPUT
END_VAR
VAR
END_VAR

METHOD OnExecute
IF NOT _ctx.hmi.bDisable THEN
	_ctx.state.iMgr.Request(_ctx.state.iIdle);
END_IF
END_METHOD

METHOD OnInit
_ctx.io.bOpenValves := TRUE;

_ctx.priv.bActive := FALSE;
_ctx.priv.bReady := FALSE;

_ctx.hmi.sStatusText := 'ROOM DISABLED!';
_ctx.hmi.nStatusColor := COL.RED.Raw;

_ctx.hmi.bHideReset := TRUE;
END_METHOD

END_FUNCTION_BLOCK

// ---- Room/State/Room_State.TcPOU
FUNCTION_BLOCK ABSTRACT Room_State EXTENDS State
VAR
	_ctx	: REFERENCE TO Room_Ctx;
END_VAR

(*FB_Init is always available implicitly and it is used primarily for initialization.
The return value is not evaluated. For a specific influence, you can also declare the
methods explicitly and provide additional code there with the standard initialization
code. You can evaluate the return value.*)
METHOD FB_Init : BOOL
VAR_INPUT
	(* TRUE: the retain variables are initialized (reset warm / reset cold)*)
	bInitRetains	: BOOL;
	(* TRUE: the instance will be copied to the copy code afterward (online change)*)
	bInCopyCode	: BOOL;
	iEntity	: Core.I_Entity;
	ctx		: REFERENCE TO Room_Ctx;
END_VAR
_ctx REF= ctx;
END_METHOD

END_FUNCTION_BLOCK

// ---- Room/State/Room_State_Fault.TcPOU
FUNCTION_BLOCK Room_State_Fault EXTENDS Room_State
VAR_INPUT
END_VAR
VAR_OUTPUT
END_VAR
VAR
END_VAR

END_FUNCTION_BLOCK

// ---- Room/State/Room_State_Idle.TcPOU
FUNCTION_BLOCK Room_State_Idle EXTENDS Room_State
VAR_INPUT
END_VAR
VAR_OUTPUT
END_VAR
VAR
END_VAR

METHOD OnExecute
IF _ctx.hmi.bDisable THEN
	_ctx.state.iMgr.Request(_ctx.state.iDisable);
END_IF
END_METHOD

METHOD OnInit
_ctx.io.bOpenValves := FALSE;

_ctx.priv.bActive := FALSE;
_ctx.priv.bReady := FALSE;

_ctx.hmi.sStatusText := 'Heating ON: Idle';
_ctx.hmi.nStatusColor := COL.BLACK.Raw;

_ctx.hmi.bHideReset := FALSE;
END_METHOD

END_FUNCTION_BLOCK

// ---- Room/State/Room_State_SystemOff.TcPOU
FUNCTION_BLOCK Room_State_SystemOff EXTENDS Room_State
VAR_INPUT
END_VAR
VAR_OUTPUT
END_VAR
VAR
END_VAR

METHOD CanDeactivate : BOOL
CanDeactivate := _ctx.priv.bSysOff;
END_METHOD

METHOD OnInit
_ctx.io.bOpenValves := FALSE;

_ctx.priv.bActive := FALSE;
_ctx.priv.bReady := FALSE;

_ctx.hmi.sStatusText := 'Central Heating is OFF';
_ctx.hmi.nStatusColor := COL.RED.Raw;

_ctx.hmi.bHideReset := FALSE;
END_METHOD

END_FUNCTION_BLOCK

// ---- Room/State/Room_State_DemandTime.TcPOU
FUNCTION_BLOCK Room_State_DemandTime EXTENDS Room_State IMPLEMENTS I_Execute
VAR
	_exe				: Execute(THIS^);
	_refTimeSettings	: REFERENCE TO Room_Settings_TimeSettings;
	_tonOff				: TON;
	_tonOn				: TON;
	
	_onRequest				: Signal;
END_VAR

METHOD CanActivate : BOOL
CanActivate := _ctx.state.iMgr.Current = _ctx.state.iIdle;
END_METHOD

METHOD Execute
VAR
	_iSelf		: I_State := THIS^;
END_VAR
IF _ctx.state.iMgr.Current <> _ctx.state.iIdle THEN
	RETURN;
END_IF

IF _ctx.state.iMgr.Current = _iSelf THEN
	_tonOff(IN := FALSE);
	RETURN;
ELSE
	_tonOff(IN := TRUE, PT := UDINT_TO_TIME(_refTimeSettings.nOff));
END_IF

IF _tonOff.Q THEN
	_tonOff(IN := FALSE);
	_ctx.state.iMgr.Request(THIS^);
END_IF
END_METHOD

(*FB_Init is always available implicitly and it is used primarily for initialization.
The return value is not evaluated. For a specific influence, you can also declare the
methods explicitly and provide additional code there with the standard initialization
code. You can evaluate the return value.*)
METHOD FB_Init : BOOL
VAR_INPUT
	(* TRUE: the retain variables are initialized (reset warm / reset cold)*)
	bInitRetains	: BOOL;
	(* TRUE: the instance will be copied to the copy code afterward (online change)*)
	bInCopyCode	: BOOL;
	iEntity	: Core.I_Entity;
	ctx			: REFERENCE TO Room_Ctx;
	refSettings		: REFERENCE TO Room_Settings_TimeSettings;
END_VAR
_refTimeSettings REF= refSettings;
END_METHOD

METHOD Init
VAR
	i			: Iter(1);
	_iEntity	: I_Entity;
	_iRec		: I_Receiver;
	_r			: Result;
	strb		: Strb;
END_VAR
WHILE IsOk(GetEntity(i.Next(), iEntity => _iEntity)) DO
	IF IsNone(GetTagOpt(_iEntity, 'Heating')) THEN
		CONTINUE;
	END_IF
	
	IF IsOk(GetReceiver(_iEntity, '*._requestRec', iRec => _iRec)) THEN
		IF IsErr(_onRequest.Pair(_iRec), nOut => _r) THEN
			DebugMsg(_iRec, strb.Append('Cannot pair _onRequest with this receiver! Error code: ').Append(TO_STRING(_r)).Read());
		END_IF
		
		EXIT;
	END_IF
END_WHILE

DebugMsg(THIS^, strb.Append('Cannot pair _systemRec with a ').Append('_requestRec').Append('!').Read());
DebugMsg(_iEntity, strb.Append('_requestRec').Append(' not found!').Read());
END_METHOD

METHOD OnExecute
_tonOn(IN := TRUE, PT := UDINT_TO_TIME(_refTimeSettings.nOn));
IF _ctx.hmi.bDisable THEN
	_ctx.state.iMgr.Request(_ctx.state.iDisable);
ELSIF _tonOn.Q THEN
	_ctx.priv.bReady := TRUE;
END_IF
END_METHOD

METHOD OnInit
_ctx.io.bOpenValves := FALSE;

_ctx.priv.bActive := TRUE;
_ctx.priv.bReady := FALSE;

_ctx.hmi.sStatusText := 'Heating ON: Scheduled demand...';
_ctx.hmi.nStatusColor := COL.BLACK.Raw;

_ctx.hmi.bHideReset := TRUE;

_tonOn(IN := FALSE);

_onRequest.Emit(_ctx.priv.iThisRoom);
END_METHOD

END_FUNCTION_BLOCK

// ---- Room/State/Room_State_DemandTemperature.TcPOU
FUNCTION_BLOCK Room_State_DemandTemperature EXTENDS Room_State IMPLEMENTS I_Execute, I_Init
VAR
	_init					: Init(THIS^);
	_exe					: Execute(THIS^);
	_refTemperatureSettings	: REFERENCE TO Room_Settings_TemperatureSettings;
	_refTemperature			: REFERENCE TO REAL;
	
	_onRequest				: Signal;
END_VAR

METHOD CanActivate : BOOL
CanActivate := _ctx.state.iMgr.Current = _ctx.state.iIdle;
END_METHOD

METHOD Execute
VAR
	_iSelf		: I_State := THIS^;
END_VAR
IF _ctx.state.iMgr.Current <> _ctx.state.iIdle THEN
	RETURN;
END_IF

IF _ctx.state.iMgr.Current = _iSelf THEN
	RETURN;
END_IF

IF _refTemperature < _refTemperatureSettings.rLow THEN
	_ctx.state.iMgr.Request(THIS^);
END_IF
END_METHOD

(*FB_Init is always available implicitly and it is used primarily for initialization.
The return value is not evaluated. For a specific influence, you can also declare the
methods explicitly and provide additional code there with the standard initialization
code. You can evaluate the return value.*)
METHOD FB_Init : BOOL
VAR_INPUT
	(* TRUE: the retain variables are initialized (reset warm / reset cold)*)
	bInitRetains	: BOOL;
	(* TRUE: the instance will be copied to the copy code afterward (online change)*)
	bInCopyCode	: BOOL;
	iEntity			: Core.I_Entity;
	ctx			: REFERENCE TO Room_Ctx;
	refSettings		: REFERENCE TO Room_Settings_TemperatureSettings;
	refTemperature	: REFERENCE TO REAL;
END_VAR
_refTemperature REF= refTemperature;
_refTemperatureSettings REF= refSettings;
END_METHOD

METHOD Init
VAR
	i			: Iter(1);
	_iEntity	: I_Entity;
	_iRec		: I_Receiver;
	_r			: Result;
	strb		: Strb;
END_VAR
WHILE IsOk(GetEntity(i.Next(), iEntity => _iEntity)) DO
	IF IsNone(GetTagOpt(_iEntity, 'Heating')) THEN
		CONTINUE;
	END_IF
	
	IF IsOk(GetReceiver(_iEntity, '*._requestRec', iRec => _iRec)) THEN
		IF IsErr(_onRequest.Pair(_iRec), nOut => _r) THEN
			DebugMsg(_iRec, strb.Append('Cannot pair _onRequest with this receiver! Error code: ').Append(TO_STRING(_r)).Read());
		END_IF
		
		EXIT;
	END_IF
END_WHILE

DebugMsg(THIS^, strb.Append('Cannot pair _systemRec with a ').Append('_requestRec').Append('!').Read());
DebugMsg(_iEntity, strb.Append('_requestRec').Append(' not found!').Read());
END_METHOD

METHOD OnExecute
IF _ctx.hmi.bDisable THEN
	_ctx.state.iMgr.Request(_ctx.state.iDisable);
ELSIF _refTemperature >= _refTemperatureSettings.rHigh THEN
	_ctx.priv.bReady := TRUE;
END_IF
END_METHOD

METHOD OnInit
_ctx.io.bOpenValves := FALSE;

_ctx.priv.bActive := TRUE;
_ctx.priv.bReady := FALSE;

_ctx.hmi.sStatusText := 'Heating ON: Low Temperature...';
_ctx.hmi.nStatusColor := COL.BLACK.Raw;

_ctx.hmi.bHideReset := TRUE;

_onRequest.Emit(_ctx.priv.iThisRoom);
END_METHOD

END_FUNCTION_BLOCK

// ---- Room/Rooms/PassiveRoom/PassiveRoom.TcPOU
FUNCTION_BLOCK PassiveRoom IMPLEMENTS I_Execute
VAR CONSTANT
	STATE_CAP		: UDINT := 5;
END_VAR
VAR
	_this			: Entity;
	_ctx			: Room_Ctx;
	_room			: RoomInterface(_ctx);
	_tag			: Tag(CONCAT('Room_', UDINT_TO_STRING(_room.Id)));
	_compTag		: Comp(_tag, _this);
	_exe			: Execute(THIS^);
	
	_uiLogic		: Room_UiLogic(_ctx);
	
	_systemReceiver	: Room_SystemReceiver(_ctx);
	
	_smgr			: StateManager<STATE_CAP>(_this);
	_proxSmgr		: StateManagerProxy(_smgr, _ctx.state.iMgr);
	
	_disable		: Room_State_Disabled(_this, _ctx);
	_proxDisable	: StateProxy(_disable, _ctx.state.iDisable);
	
	_fault			: Room_State_Fault(_this,_ctx);
	_proxFault		: StateProxy(_fault, _ctx.state.iFault);	
	
	_idle			: Room_State_Idle(_this,_ctx);
	_proxIdle		: StateProxy(_idle, _ctx.state.iIdle);	
	
	_systemOff		: Room_State_SystemOff(_this,_ctx);
	_proxSystemOff	: StateProxy(_systemOff, _ctx.state.iSystemOff);
END_VAR

// Here add custom components

VAR PERSISTENT
	_bEnablePassive	: BOOL;
END_VAR
VAR_INPUT
	bInletValveIsOpen		: BOOL;
	bInletValveIsClosed		: BOOL;
	
	bOutletValveIsOpen		: BOOL;
	bOutletValveIsClosed	: BOOL;
END_VAR
VAR_OUTPUT
	bInletValve			: BOOL;
	bOutletValve		: BOOL;
END_VAR
VAR
	_passiveDemand	: Room_State_DemandPassive(_this, _ctx, _bEnablePassive);
END_VAR

METHOD Execute
_ctx.priv.bClosed := bInletValveIsClosed AND bOutletValveIsClosed;
_ctx.priv.bOpen := bInletValveIsOpen AND bOutletValveIsOpen;

bInletValve :=  _ctx.io.bOpenValves;
bOutletValve :=  _ctx.io.bOpenValves;
END_METHOD

END_FUNCTION_BLOCK

// ---- Room/State/Room_State_DemandPassive.TcPOU
FUNCTION_BLOCK Room_State_DemandPassive EXTENDS Room_State IMPLEMENTS I_Execute, I_Init
VAR
	_init					: Init(THIS^);
	_exe					: Execute(THIS^);
	_refEnable				: REFERENCE TO BOOL;
	_onPassiveStateChange	: Signal;
	_bIsPassive				: BoolArg;
END_VAR

METHOD CanActivate : BOOL
CanActivate := _ctx.state.iMgr.Current = _ctx.state.iIdle;
END_METHOD

METHOD Execute
VAR
	_iSelf		: I_State := THIS^;
END_VAR
IF _ctx.state.iMgr.Current <> _ctx.state.iIdle THEN
	RETURN;
END_IF

IF _ctx.state.iMgr.Current = _iSelf THEN
	RETURN;
END_IF

IF _refEnable AND NOT _ctx.priv.bPaused THEN
	_ctx.state.iMgr.Request(THIS^);
END_IF
END_METHOD

(*FB_Init is always available implicitly and it is used primarily for initialization.
The return value is not evaluated. For a specific influence, you can also declare the
methods explicitly and provide additional code there with the standard initialization
code. You can evaluate the return value.*)
METHOD FB_Init : BOOL
VAR_INPUT
	(* TRUE: the retain variables are initialized (reset warm / reset cold)*)
	bInitRetains	: BOOL;
	(* TRUE: the instance will be copied to the copy code afterward (online change)*)
	bInCopyCode	: BOOL;
	iEntity	: Core.I_Entity;
	ctx			: REFERENCE TO Room_Ctx;
	refEnable	: REFERENCE TO BOOL;
END_VAR
_refEnable REF= refEnable;
END_METHOD

METHOD Init
VAR
	i			: Iter(1);
	_iEntity	: I_Entity;
	_iRec		: I_Receiver;
	_r			: Result;
	strb		: Strb;
END_VAR
WHILE IsOk(GetEntity(i.Next(), iEntity => _iEntity)) DO
	IF IsNone(GetTagOpt(_iEntity, 'Heating')) THEN
		CONTINUE;
	END_IF
	
	IF IsOk(GetReceiver(_iEntity, '*._passiveHeatingCountRec', iRec => _iRec)) THEN
		IF IsErr(_onPassiveStateChange.Pair(_iRec), nOut => _r) THEN
			DebugMsg(_iRec, strb.Append('Cannot pair _onPassiveStateChange with this receiver! Error code: ').Append(TO_STRING(_r)).Read());
		END_IF
		
		RETURN;
	END_IF
END_WHILE
END_METHOD

METHOD OnExecute
IF _ctx.hmi.bDisable THEN	
	_ctx.state.iMgr.Request(_ctx.state.iDisable);
ELSIF _refEnable THEN
	_ctx.state.iMgr.Request(_ctx.state.iIdle);
ELSIF _ctx.priv.bPaused THEN
	_ctx.state.iMgr.Request(_ctx.state.iIdle);
END_IF
END_METHOD

METHOD OnExit
_bIsPassive.Val := FALSE;
_onPassiveStateChange.Emit(_bIsPassive);
END_METHOD

METHOD OnInit
_ctx.io.bOpenValves := TRUE;

_ctx.priv.bActive := TRUE;
_ctx.priv.bReady := FALSE;

_ctx.hmi.sStatusText := 'Heating ON: Passive mode...';
_ctx.hmi.nStatusColor := COL.BLACK.Raw;

_ctx.hmi.bHideReset := TRUE;

_bIsPassive.Val := TRUE;
_onPassiveStateChange.Emit(_bIsPassive);
END_METHOD

END_FUNCTION_BLOCK

// ---- Room/Rooms/FullRoom/PassiveTempTimeRoom.TcPOU
FUNCTION_BLOCK PassiveTempTimeRoom IMPLEMENTS I_Execute
VAR CONSTANT
	STATE_CAP		: UDINT := 7;
END_VAR
VAR
	_this			: Entity;
	_ctx			: Room_Ctx;
	_room			: RoomInterface(_ctx);
	_tag			: Tag(CONCAT('Room_', UDINT_TO_STRING(_room.Id)));
	_compTag		: Comp(_tag, _this);
	_exe			: Execute(THIS^);
	
	_uiLogic		: Room_UiLogic(_ctx);
	
	_systemReceiver	: Room_SystemReceiver(_ctx);
	
	_smgr			: StateManager<STATE_CAP>(_this);
	_proxSmgr		: StateManagerProxy(_smgr, _ctx.state.iMgr);
	
	_disable		: Room_State_Disabled(_this, _ctx);
	_proxDisable	: StateProxy(_disable, _ctx.state.iDisable);
	
	_fault			: Room_State_Fault(_this,_ctx);
	_proxFault		: StateProxy(_fault, _ctx.state.iFault);	
	
	_idle			: Room_State_Idle(_this,_ctx);
	_proxIdle		: StateProxy(_idle, _ctx.state.iIdle);	
	
	_systemOff		: Room_State_SystemOff(_this,_ctx);
	_proxSystemOff	: StateProxy(_systemOff, _ctx.state.iSystemOff);
END_VAR

// Here add custom components

VAR PERSISTENT
	_settings		: Room_Settings_PassiveTempTime;
END_VAR

VAR_INPUT
	rTemperature	: REAL;

	bInletValveIsOpen		: BOOL;
	bInletValveIsClosed		: BOOL;
	
	bOutletValveIsOpen		: BOOL;
	bOutletValveIsClosed	: BOOL;
END_VAR
VAR_OUTPUT
	bInletValve			: BOOL;
	bOutletValve		: BOOL;
END_VAR
VAR
	_timeDemand		: Room_State_DemandTime(_this, _ctx, _settings.timee);
	_tempDemand		: Room_State_DemandTemperature(_this, _ctx, _settings.temp, rTemperature);
	_passiveDemand	: Room_State_DemandPassive(_this, _ctx, _settings.bEnablePassive);
END_VAR

METHOD Execute
_ctx.priv.bClosed := bInletValveIsClosed AND bOutletValveIsClosed;
_ctx.priv.bOpen := bInletValveIsOpen AND bOutletValveIsOpen;

bInletValve :=  _ctx.io.bOpenValves;
bOutletValve :=  _ctx.io.bOpenValves;
END_METHOD

END_FUNCTION_BLOCK

// ---- Room/Rooms/FullRoom/PassiveTempTimeRoomWithMultipleValves.TcPOU
FUNCTION_BLOCK PassiveTempTimeRoomWithMultipleValves 
VAR_GENERIC CONSTANT
	VALVE_CAP		: UDINT := 7;
END_VAR

IMPLEMENTS I_Execute

VAR CONSTANT
	STATE_CAP		: UDINT := 7;
END_VAR
VAR
	_this			: Entity;
	_ctx			: Room_Ctx;
	_room			: RoomInterface(_ctx);
	_tag			: Tag(CONCAT('Room_', UDINT_TO_STRING(_room.Id)));
	_compTag		: Comp(_tag, _this);
	_exe			: Execute(THIS^);
	
	_uiLogic		: Room_UiLogic(_ctx);
	
	_systemReceiver	: Room_SystemReceiver(_ctx);
	
	_smgr			: StateManager<STATE_CAP>(_this);
	_proxSmgr		: StateManagerProxy(_smgr, _ctx.state.iMgr);
	
	_disable		: Room_State_Disabled(_this, _ctx);
	_proxDisable	: StateProxy(_disable, _ctx.state.iDisable);
	
	_fault			: Room_State_Fault(_this,_ctx);
	_proxFault		: StateProxy(_fault, _ctx.state.iFault);	
	
	_idle			: Room_State_Idle(_this,_ctx);
	_proxIdle		: StateProxy(_idle, _ctx.state.iIdle);	
	
	_systemOff		: Room_State_SystemOff(_this,_ctx);
	_proxSystemOff	: StateProxy(_systemOff, _ctx.state.iSystemOff);
END_VAR

// Here add custom components

VAR PERSISTENT
	_settings		: Room_Settings_PassiveTempTime;
END_VAR
VAR_INPUT
	rTemperature	: REAL;

	bInletValveIsOpen		: BOOL;
	bInletValveIsClosed		: BOOL;
	
	bOutletValveIsOpen		: ARRAY[1..VALVE_CAP] OF BOOL;
	bOutletValveIsClosed	: ARRAY[1..VALVE_CAP] OF BOOL;
END_VAR
VAR_OUTPUT
	bInletValve			: ARRAY[1..VALVE_CAP] OF BOOL;
	bOutletValve		: ARRAY[1..VALVE_CAP] OF BOOL;
END_VAR
VAR
	_timeDemand		: Room_State_DemandTime(_this, _ctx, _settings.timee);
	_tempDemand		: Room_State_DemandTemperature(_this, _ctx, _settings.temp, rTemperature);
	_passiveDemand	: Room_State_DemandPassive(_this, _ctx, _settings.bEnablePassive);
END_VAR

METHOD Execute
VAR
	i			: UDINT;
END_VAR
_ctx.priv.bClosed := TRUE;
_ctx.priv.bOpen := TRUE;

FOR i := 1 TO VALVE_CAP DO
	bInletValve[i] :=  _ctx.io.bOpenValves;
	bOutletValve[i] :=  _ctx.io.bOpenValves;	
	
	_ctx.priv.bClosed := _ctx.priv.bClosed AND bOutletValveIsClosed[i];
	_ctx.priv.bOpen := _ctx.priv.bClosed AND bOutletValveIsOpen[i];	
END_FOR
END_METHOD

END_FUNCTION_BLOCK

// ---- Room/Rooms/TempRoom/TempRoom.TcPOU
FUNCTION_BLOCK TempRoom IMPLEMENTS I_Execute
VAR CONSTANT
	STATE_CAP		: UDINT := 5;
END_VAR
VAR
	_this			: Entity;
	_ctx			: Room_Ctx;
	_room			: RoomInterface(_ctx);
	_tag			: Tag(CONCAT('Room_', UDINT_TO_STRING(_room.Id)));
	_compTag		: Comp(_tag, _this);
	_exe			: Execute(THIS^);
	
	_uiLogic		: Room_UiLogic(_ctx);
	
	_systemReceiver	: Room_SystemReceiver(_ctx);
	
	_smgr			: StateManager<STATE_CAP>(_this);
	_proxSmgr		: StateManagerProxy(_smgr, _ctx.state.iMgr);
	
	_disable		: Room_State_Disabled(_this, _ctx);
	_proxDisable	: StateProxy(_disable, _ctx.state.iDisable);
	
	_fault			: Room_State_Fault(_this,_ctx);
	_proxFault		: StateProxy(_fault, _ctx.state.iFault);	
	
	_idle			: Room_State_Idle(_this,_ctx);
	_proxIdle		: StateProxy(_idle, _ctx.state.iIdle);	
	
	_systemOff		: Room_State_SystemOff(_this,_ctx);
	_proxSystemOff	: StateProxy(_systemOff, _ctx.state.iSystemOff);
END_VAR

	// Here add custom components

VAR PERSISTENT
	_settings				: Room_Settings_TemperatureSettings;
END_VAR
VAR_INPUT
	rTemperature			: REAL;
	
	bInletValveIsOpen		: BOOL;
	bInletValveIsClosed		: BOOL;
	
	bOutletValveIsOpen		: BOOL;
	bOutletValveIsClosed	: BOOL;
END_VAR

VAR_OUTPUT
	bInletValve				: BOOL;
	bOutletValve			: BOOL;
END_VAR
VAR
	_tempDemand		: Room_State_DemandTemperature(_this, _ctx, _settings, rTemperature);
END_VAR

METHOD Execute
VAR
	i			: UDINT;
	_rTempSum	: REAL;
END_VAR
_ctx.priv.bClosed := bInletValveIsClosed AND bOutletValveIsClosed;
_ctx.priv.bOpen := bInletValveIsOpen AND bOutletValveIsOpen;

bInletValve :=  _ctx.io.bOpenValves;
bOutletValve :=  _ctx.io.bOpenValves;
END_METHOD

END_FUNCTION_BLOCK

// ---- Room/Rooms/TempRoom/TempRoomWithMultipleSensors.TcPOU
FUNCTION_BLOCK TempRoomWithMultipleSensors
VAR_GENERIC CONSTANT
	SENSOR_CAP		: UDINT := 4;
END_VAR
IMPLEMENTS I_Execute
VAR CONSTANT
	STATE_CAP		: UDINT := 5;
END_VAR
VAR
	_this			: Entity;
	_ctx			: Room_Ctx;
	_room			: RoomInterface(_ctx);
	_tag			: Tag(CONCAT('Room_', UDINT_TO_STRING(_room.Id)));
	_compTag		: Comp(_tag, _this);
	_exe			: Execute(THIS^);
	
	_uiLogic		: Room_UiLogic(_ctx);
	
	_systemReceiver	: Room_SystemReceiver(_ctx);
	
	_smgr			: StateManager<STATE_CAP>(_this);
	_proxSmgr		: StateManagerProxy(_smgr, _ctx.state.iMgr);
	
	_disable		: Room_State_Disabled(_this, _ctx);
	_proxDisable	: StateProxy(_disable, _ctx.state.iDisable);
	
	_fault			: Room_State_Fault(_this,_ctx);
	_proxFault		: StateProxy(_fault, _ctx.state.iFault);	
	
	_idle			: Room_State_Idle(_this,_ctx);
	_proxIdle		: StateProxy(_idle, _ctx.state.iIdle);	
	
	_systemOff		: Room_State_SystemOff(_this,_ctx);
	_proxSystemOff	: StateProxy(_systemOff, _ctx.state.iSystemOff);
END_VAR

	// Here add custom components

VAR PERSISTENT
	_settings				: Room_Settings_TemperatureSettings;
END_VAR
VAR_INPUT
	rTemperature			: ARRAY[1..SENSOR_CAP] OF REAL;
	
	bInletValveIsOpen		: BOOL;
	bInletValveIsClosed		: BOOL;
	
	bOutletValveIsOpen		: BOOL;
	bOutletValveIsClosed	: BOOL;
END_VAR
VAR
	_rTemperature			: REAL;
END_VAR
VAR_OUTPUT
	bInletValve				: BOOL;
	bOutletValve			: BOOL;
END_VAR
VAR
	_tempDemand		: Room_State_DemandTemperature(_this, _ctx, _settings, _rTemperature);
END_VAR

METHOD Execute
VAR
	i			: UDINT;
	_rTempSum	: REAL;
END_VAR
_ctx.priv.bClosed := bInletValveIsClosed AND bOutletValveIsClosed;
_ctx.priv.bOpen := bInletValveIsOpen AND bOutletValveIsOpen;

bInletValve :=  _ctx.io.bOpenValves;
bOutletValve :=  _ctx.io.bOpenValves;

FOR i := 1 TO SENSOR_CAP DO
	_rTempSum := rTemperature[i] + _rTempSum;
END_FOR

_rTemperature := _rTempSum/UDINT_TO_REAL(SENSOR_CAP);
END_METHOD

END_FUNCTION_BLOCK

// ---- Room/Rooms/TimeRoom/TimeRoom.TcPOU
FUNCTION_BLOCK TimeRoom IMPLEMENTS I_Execute
VAR CONSTANT
	STATE_CAP		: UDINT := 5;
END_VAR
VAR
	_this			: Entity;
	_ctx			: Room_Ctx;
	_room			: RoomInterface(_ctx);
	_tag			: Tag(CONCAT('Room_', UDINT_TO_STRING(_room.Id)));
	_compTag		: Comp(_tag, _this);
	_exe			: Execute(THIS^);
	
	_uiLogic		: Room_UiLogic(_ctx);
	
	_systemReceiver	: Room_SystemReceiver(_ctx);
	
	_smgr			: StateManager<STATE_CAP>(_this);
	_proxSmgr		: StateManagerProxy(_smgr, _ctx.state.iMgr);
	
	_disable		: Room_State_Disabled(_this, _ctx);
	_proxDisable	: StateProxy(_disable, _ctx.state.iDisable);
	
	_fault			: Room_State_Fault(_this,_ctx);
	_proxFault		: StateProxy(_fault, _ctx.state.iFault);	
	
	_idle			: Room_State_Idle(_this,_ctx);
	_proxIdle		: StateProxy(_idle, _ctx.state.iIdle);	
	
	_systemOff		: Room_State_SystemOff(_this,_ctx);
	_proxSystemOff	: StateProxy(_systemOff, _ctx.state.iSystemOff);
END_VAR

	// Here add custom components

VAR PERSISTENT
	_settings		: Room_Settings_TimeSettings;
END_VAR
VAR_INPUT
	bInletValveIsOpen		: BOOL;
	bInletValveIsClosed		: BOOL;
	
	bOutletValveIsOpen		: BOOL;
	bOutletValveIsClosed	: BOOL;
END_VAR
VAR_OUTPUT
	bInletValve			: BOOL;
	bOutletValve		: BOOL;
END_VAR
VAR
	_timeDemand		: Room_State_DemandTime(_this, _ctx, _settings);
END_VAR

METHOD Execute
_ctx.priv.bClosed := bInletValveIsClosed AND bOutletValveIsClosed;
_ctx.priv.bOpen := bInletValveIsOpen AND bOutletValveIsOpen;

bInletValve :=  _ctx.io.bOpenValves;
bOutletValve :=  _ctx.io.bOpenValves;
END_METHOD

END_FUNCTION_BLOCK

// ---- Room/Rooms/AbstractRoom.TcPOU
// THIS SHOULD BE COPIED AND NOT EXTENDED!!!
FUNCTION_BLOCK ABSTRACT AbstractRoom IMPLEMENTS I_Execute
VAR CONSTANT
	STATE_CAP		: UDINT := 4;
END_VAR
VAR
	_this			: Entity;
	_ctx			: Room_Ctx;
	_room			: RoomInterface(_ctx);
	_tag			: Tag(CONCAT('Room_', UDINT_TO_STRING(_room.Id)));
	_compTag		: Comp(_tag, _this);
	_exe			: Execute(THIS^);
	
	_uiLogic		: Room_UiLogic(_ctx);
	
	_systemReceiver	: Room_SystemReceiver(_ctx);
	
	_smgr			: StateManager<STATE_CAP>(_this);
	_proxSmgr		: StateManagerProxy(_smgr, _ctx.state.iMgr);
	
	_disable		: Room_State_Disabled(_this, _ctx);
	_proxDisable	: StateProxy(_disable, _ctx.state.iDisable);
	
	_fault			: Room_State_Fault(_this,_ctx);
	_proxFault		: StateProxy(_fault, _ctx.state.iFault);	
	
	_idle			: Room_State_Idle(_this,_ctx);
	_proxIdle		: StateProxy(_idle, _ctx.state.iIdle);	
	
	_systemOff		: Room_State_SystemOff(_this,_ctx);
	_proxSystemOff	: StateProxy(_systemOff, _ctx.state.iSystemOff);
END_VAR

	// Here add custom components

METHOD Execute
END_METHOD

END_FUNCTION_BLOCK

// ---- GlobalTextList.TcGTLO
TEXTLIST GlobalTextList
  443 = '%.2f'
  862 = '%s'
  553 = 'Auto Sim'
  870 = 'Click to change'
  969 = 'Drain Outlet Open'
  754 = 'Drain Outlet Valve Open'
  445 = 'Drain Speed: %.4f'
  336 = 'Enable Switch'
  958 = 'Enable Tank Switch'
  520 = 'EStop Button'
  707 = 'Feedback Ok'
  476 = 'Fill Speed: %.4f'
  923 = 'Filling Timeout:'
  698 = 'Filling Timeout: %s'
  371 = 'High Level: %.2f'
  140 = 'High Level: %s'
  254 = 'hmi.sMultiButtonText'
  89 = 'Level Sensor'
  616 = 'Low Level: %.2f'
  234 = 'Low Level: %s'
  700 = 'NoWater'
  998 = 'Overload'
  116 = 'Press to Reset'
  342 = 'Pump'
  190 = 'Request Button'
  261 = 'Request Level: %.2f'
  452 = 'Request Level: %s'
  160 = 'Reset Output'
  305 = 'Run Output'
  300 = 'RunPump'
  629 = 'Simulation'
  411 = 'State:'
  587 = 'State: %s'
  664 = 'Status:'
  338 = 'System Operational'
  12 = 'Tank 0'
  237 = 'Tank 1'
  741 = 'Tank 2'
  288 = 'Tank 3'
  737 = 'Timeout: %.2f'
  430 = 'Timeout: %s'
END_TEXTLIST
